(* CoDeSys 2.3 export: MNG_RAWDATAGRAM.EXP *)

(* Data type in MNG_TCPIP *)
TYPE MNG_RawDatagram :(* binary TCP/IP datagram (4 byte aligned) *)
STRUCT
	Header	:  MNG_DatagramHeader;(* datagram header *)
	Payload	:  MNG_DataARRAY;
END_STRUCT
END_TYPE
